// TIA Portal V18 export
TYPE "UDT_settingsSirene"
// stored: IsFailsafeCompliant false
   STRUCT
      toneSelect { ExternalVisible := 'False'; S7_SetPoint := 'True'} : DInt;
      toneDuration { ExternalVisible := 'False'; S7_SetPoint := 'True'} : Time;
      test { ExternalVisible := 'False'; S7_SetPoint := 'True'} : DInt;
   END_STRUCT;
END_TYPE
